// TIA Portal V19 export
FUNCTION "AO SCALING" : Void   // FC13, LAD
{ S7_Optimized_Access := 'TRUE' }
// stored: SetENOAutomatically false
BEGIN

REGION Network 1: VFD P-502A
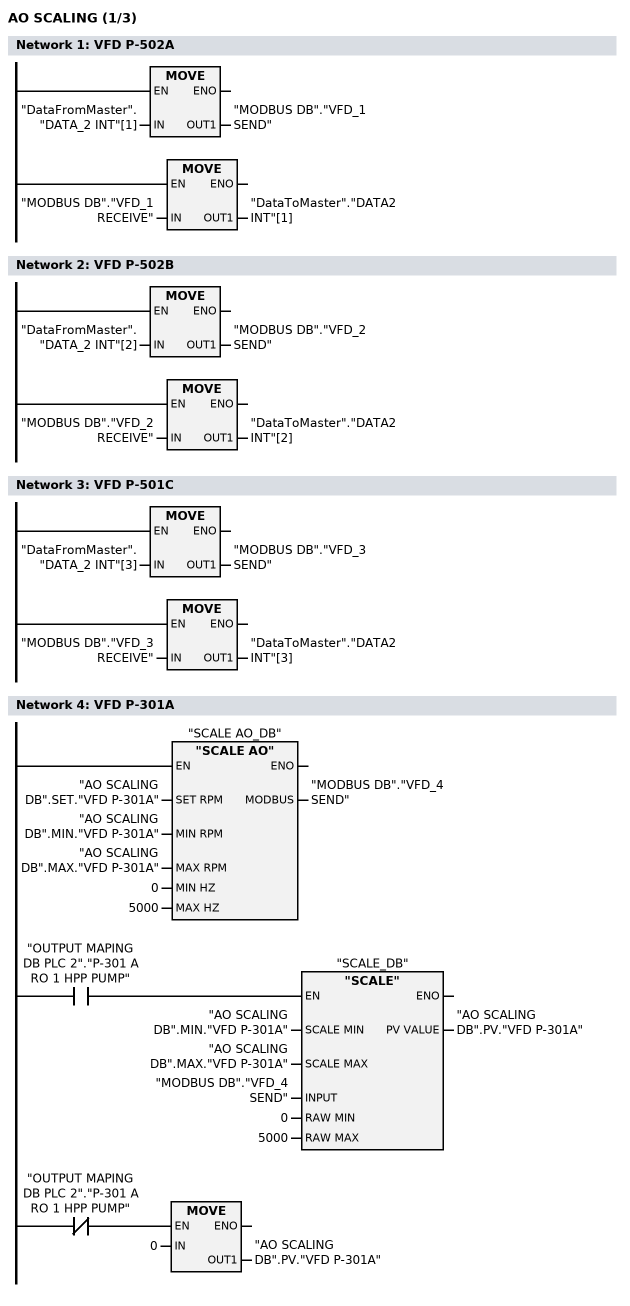
   RUNG wire#powerrail
      Move(in := "DataFromMaster"."DATA_2 INT"[1], out1 => "MODBUS DB"."VFD_1 SEND")
   END_RUNG
   RUNG wire#powerrail
      Move(in := "MODBUS DB"."VFD_1 RECEIVE", out1 => "DataToMaster"."DATA2 INT"[1])
   END_RUNG
   // the same network as SCL:
   "MODBUS DB"."VFD_1 SEND" := "DataFromMaster"."DATA_2 INT"[1];
   "DataToMaster"."DATA2 INT"[1] := "MODBUS DB"."VFD_1 RECEIVE";
END_REGION

REGION Network 2: VFD P-502B
   RUNG wire#powerrail
      Move(in := "DataFromMaster"."DATA_2 INT"[2], out1 => "MODBUS DB"."VFD_2 SEND")
   END_RUNG
   RUNG wire#powerrail
      Move(in := "MODBUS DB"."VFD_2 RECEIVE", out1 => "DataToMaster"."DATA2 INT"[2])
   END_RUNG
   // the same network as SCL:
   "MODBUS DB"."VFD_2 SEND" := "DataFromMaster"."DATA_2 INT"[2];
   "DataToMaster"."DATA2 INT"[2] := "MODBUS DB"."VFD_2 RECEIVE";
END_REGION

REGION Network 3: VFD P-501C
   RUNG wire#powerrail
      Move(in := "DataFromMaster"."DATA_2 INT"[3], out1 => "MODBUS DB"."VFD_3 SEND")
   END_RUNG
   RUNG wire#powerrail
      Move(in := "MODBUS DB"."VFD_3 RECEIVE", out1 => "DataToMaster"."DATA2 INT"[3])
   END_RUNG
   // the same network as SCL:
   "MODBUS DB"."VFD_3 SEND" := "DataFromMaster"."DATA_2 INT"[3];
   "DataToMaster"."DATA2 INT"[3] := "MODBUS DB"."VFD_3 RECEIVE";
END_REGION

REGION Network 4: VFD P-301A
   RUNG wire#powerrail
      "SCALE AO_DB"("SET RPM" := "AO SCALING DB".SET."VFD P-301A", "MIN RPM" := "AO SCALING DB".MIN."VFD P-301A", "MAX RPM" := "AO SCALING DB".MAX."VFD P-301A", "MIN HZ" := 0, "MAX HZ" := 5000, MODBUS => "MODBUS DB"."VFD_4 SEND")
   END_RUNG
   RUNG wire#powerrail
      Contact( "OUTPUT MAPING DB PLC 2"."P-301 A RO 1 HPP PUMP" )
      "SCALE_DB"("SCALE MIN" := "AO SCALING DB".MIN."VFD P-301A", "SCALE MAX" := "AO SCALING DB".MAX."VFD P-301A", INPUT := "MODBUS DB"."VFD_4 SEND", "RAW MIN" := 0, "RAW MAX" := 5000, "PV VALUE" => "AO SCALING DB".PV."VFD P-301A")
   END_RUNG
   RUNG wire#powerrail
      I_Contact( "OUTPUT MAPING DB PLC 2"."P-301 A RO 1 HPP PUMP" )
      Move(in := 0, out1 => "AO SCALING DB".PV."VFD P-301A")
   END_RUNG
   // the same network as SCL:
   "SCALE AO_DB"("SET RPM" := "AO SCALING DB".SET."VFD P-301A",   // "SCALE AO"
                 "MIN RPM" := "AO SCALING DB".MIN."VFD P-301A",
                 "MAX RPM" := "AO SCALING DB".MAX."VFD P-301A",
                 "MIN HZ" := 0,
                 "MAX HZ" := 5000,
                 MODBUS => "MODBUS DB"."VFD_4 SEND");
   IF "OUTPUT MAPING DB PLC 2"."P-301 A RO 1 HPP PUMP" THEN
       "SCALE_DB"("SCALE MIN" := "AO SCALING DB".MIN."VFD P-301A",   // "SCALE"
                  "SCALE MAX" := "AO SCALING DB".MAX."VFD P-301A",
                  INPUT := "MODBUS DB"."VFD_4 SEND",
                  "RAW MIN" := 0,
                  "RAW MAX" := 5000,
                  "PV VALUE" => "AO SCALING DB".PV."VFD P-301A");
   END_IF;
   IF NOT "OUTPUT MAPING DB PLC 2"."P-301 A RO 1 HPP PUMP" THEN "AO SCALING DB".PV."VFD P-301A" := 0; END_IF;
END_REGION

REGION Network 5: VFD P-301B
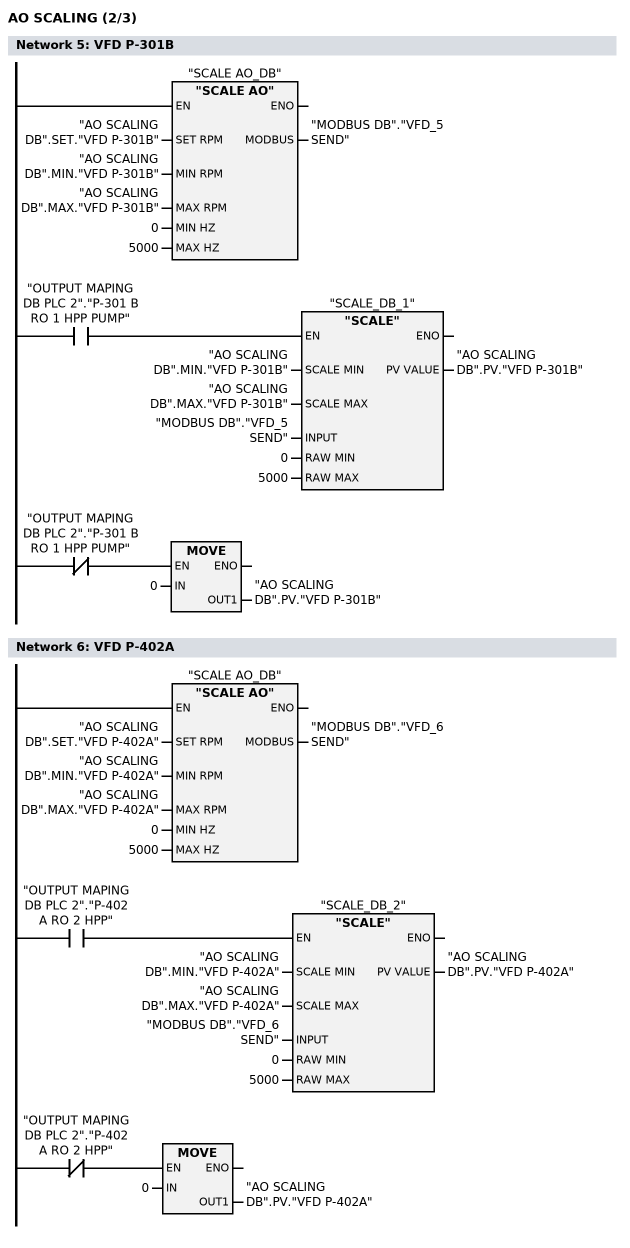
   RUNG wire#powerrail
      "SCALE AO_DB"("SET RPM" := "AO SCALING DB".SET."VFD P-301B", "MIN RPM" := "AO SCALING DB".MIN."VFD P-301B", "MAX RPM" := "AO SCALING DB".MAX."VFD P-301B", "MIN HZ" := 0, "MAX HZ" := 5000, MODBUS => "MODBUS DB"."VFD_5 SEND")
   END_RUNG
   RUNG wire#powerrail
      Contact( "OUTPUT MAPING DB PLC 2"."P-301 B RO 1 HPP PUMP" )
      "SCALE_DB_1"("SCALE MIN" := "AO SCALING DB".MIN."VFD P-301B", "SCALE MAX" := "AO SCALING DB".MAX."VFD P-301B", INPUT := "MODBUS DB"."VFD_5 SEND", "RAW MIN" := 0, "RAW MAX" := 5000, "PV VALUE" => "AO SCALING DB".PV."VFD P-301B")
   END_RUNG
   RUNG wire#powerrail
      I_Contact( "OUTPUT MAPING DB PLC 2"."P-301 B RO 1 HPP PUMP" )
      Move(in := 0, out1 => "AO SCALING DB".PV."VFD P-301B")
   END_RUNG
   // the same network as SCL:
   "SCALE AO_DB"("SET RPM" := "AO SCALING DB".SET."VFD P-301B",   // "SCALE AO"
                 "MIN RPM" := "AO SCALING DB".MIN."VFD P-301B",
                 "MAX RPM" := "AO SCALING DB".MAX."VFD P-301B",
                 "MIN HZ" := 0,
                 "MAX HZ" := 5000,
                 MODBUS => "MODBUS DB"."VFD_5 SEND");
   IF "OUTPUT MAPING DB PLC 2"."P-301 B RO 1 HPP PUMP" THEN
       "SCALE_DB_1"("SCALE MIN" := "AO SCALING DB".MIN."VFD P-301B",   // "SCALE"
                    "SCALE MAX" := "AO SCALING DB".MAX."VFD P-301B",
                    INPUT := "MODBUS DB"."VFD_5 SEND",
                    "RAW MIN" := 0,
                    "RAW MAX" := 5000,
                    "PV VALUE" => "AO SCALING DB".PV."VFD P-301B");
   END_IF;
   IF NOT "OUTPUT MAPING DB PLC 2"."P-301 B RO 1 HPP PUMP" THEN "AO SCALING DB".PV."VFD P-301B" := 0; END_IF;
END_REGION

REGION Network 6: VFD P-402A
   RUNG wire#powerrail
      "SCALE AO_DB"("SET RPM" := "AO SCALING DB".SET."VFD P-402A", "MIN RPM" := "AO SCALING DB".MIN."VFD P-402A", "MAX RPM" := "AO SCALING DB".MAX."VFD P-402A", "MIN HZ" := 0, "MAX HZ" := 5000, MODBUS => "MODBUS DB"."VFD_6 SEND")
   END_RUNG
   RUNG wire#powerrail
      Contact( "OUTPUT MAPING DB PLC 2"."P-402  A RO 2 HPP" )
      "SCALE_DB_2"("SCALE MIN" := "AO SCALING DB".MIN."VFD P-402A", "SCALE MAX" := "AO SCALING DB".MAX."VFD P-402A", INPUT := "MODBUS DB"."VFD_6 SEND", "RAW MIN" := 0, "RAW MAX" := 5000, "PV VALUE" => "AO SCALING DB".PV."VFD P-402A")
   END_RUNG
   RUNG wire#powerrail
      I_Contact( "OUTPUT MAPING DB PLC 2"."P-402  A RO 2 HPP" )
      Move(in := 0, out1 => "AO SCALING DB".PV."VFD P-402A")
   END_RUNG
   // the same network as SCL:
   "SCALE AO_DB"("SET RPM" := "AO SCALING DB".SET."VFD P-402A",   // "SCALE AO"
                 "MIN RPM" := "AO SCALING DB".MIN."VFD P-402A",
                 "MAX RPM" := "AO SCALING DB".MAX."VFD P-402A",
                 "MIN HZ" := 0,
                 "MAX HZ" := 5000,
                 MODBUS => "MODBUS DB"."VFD_6 SEND");
   IF "OUTPUT MAPING DB PLC 2"."P-402  A RO 2 HPP" THEN
       "SCALE_DB_2"("SCALE MIN" := "AO SCALING DB".MIN."VFD P-402A",   // "SCALE"
                    "SCALE MAX" := "AO SCALING DB".MAX."VFD P-402A",
                    INPUT := "MODBUS DB"."VFD_6 SEND",
                    "RAW MIN" := 0,
                    "RAW MAX" := 5000,
                    "PV VALUE" => "AO SCALING DB".PV."VFD P-402A");
   END_IF;
   IF NOT "OUTPUT MAPING DB PLC 2"."P-402  A RO 2 HPP" THEN "AO SCALING DB".PV."VFD P-402A" := 0; END_IF;
END_REGION

REGION Network 7: VFD P-402B
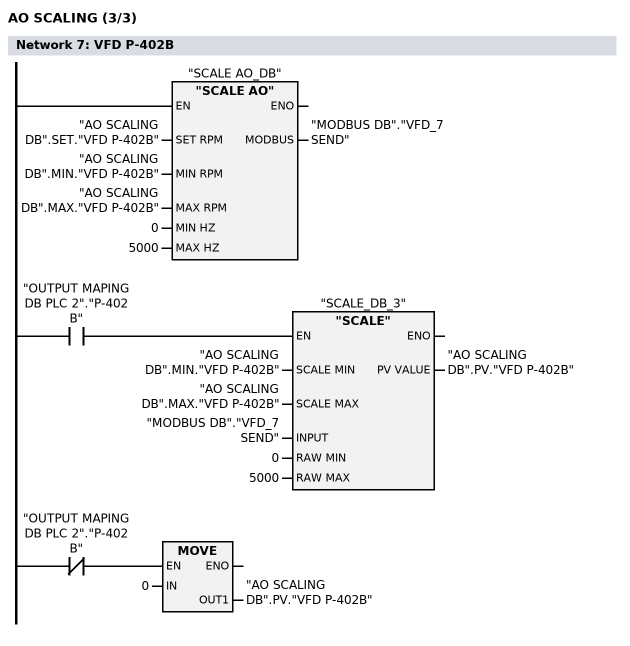
   RUNG wire#powerrail
      "SCALE AO_DB"("SET RPM" := "AO SCALING DB".SET."VFD P-402B", "MIN RPM" := "AO SCALING DB".MIN."VFD P-402B", "MAX RPM" := "AO SCALING DB".MAX."VFD P-402B", "MIN HZ" := 0, "MAX HZ" := 5000, MODBUS => "MODBUS DB"."VFD_7 SEND")
   END_RUNG
   RUNG wire#powerrail
      Contact( "OUTPUT MAPING DB PLC 2"."P-402 B" )
      "SCALE_DB_3"("SCALE MIN" := "AO SCALING DB".MIN."VFD P-402B", "SCALE MAX" := "AO SCALING DB".MAX."VFD P-402B", INPUT := "MODBUS DB"."VFD_7 SEND", "RAW MIN" := 0, "RAW MAX" := 5000, "PV VALUE" => "AO SCALING DB".PV."VFD P-402B")
   END_RUNG
   RUNG wire#powerrail
      I_Contact( "OUTPUT MAPING DB PLC 2"."P-402 B" )
      Move(in := 0, out1 => "AO SCALING DB".PV."VFD P-402B")
   END_RUNG
   // the same network as SCL:
   "SCALE AO_DB"("SET RPM" := "AO SCALING DB".SET."VFD P-402B",   // "SCALE AO"
                 "MIN RPM" := "AO SCALING DB".MIN."VFD P-402B",
                 "MAX RPM" := "AO SCALING DB".MAX."VFD P-402B",
                 "MIN HZ" := 0,
                 "MAX HZ" := 5000,
                 MODBUS => "MODBUS DB"."VFD_7 SEND");
   IF "OUTPUT MAPING DB PLC 2"."P-402 B" THEN
       "SCALE_DB_3"("SCALE MIN" := "AO SCALING DB".MIN."VFD P-402B",   // "SCALE"
                    "SCALE MAX" := "AO SCALING DB".MAX."VFD P-402B",
                    INPUT := "MODBUS DB"."VFD_7 SEND",
                    "RAW MIN" := 0,
                    "RAW MAX" := 5000,
                    "PV VALUE" => "AO SCALING DB".PV."VFD P-402B");
   END_IF;
   IF NOT "OUTPUT MAPING DB PLC 2"."P-402 B" THEN "AO SCALING DB".PV."VFD P-402B" := 0; END_IF;
END_REGION
END_FUNCTION
